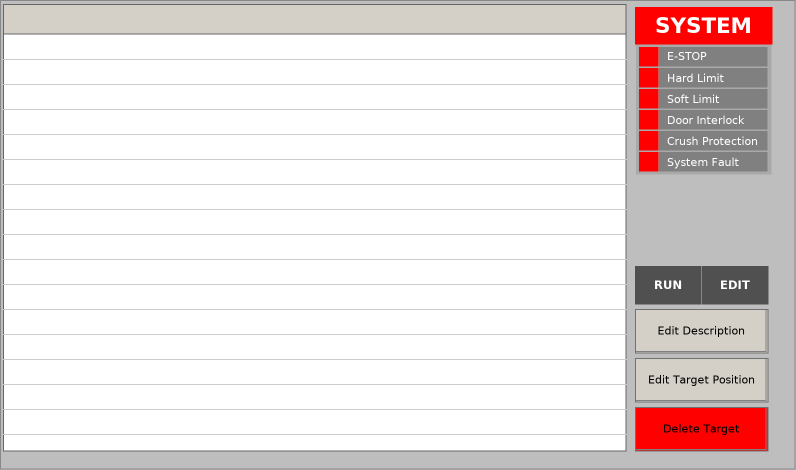
VISUALIZATION TARGET_PANEL  // 796x470
    Button (635,358 133x44), "Edit Target Position", colour toggle: (GV_HMI.ColorToggle[2])<>0, invisible if: HMI.bEditEnable<>1
        tap GV_HMI.ColorToggle[2]
        OnDialogClosed: execute {
            IF XML.savedvalues.savedpos[GV_HMI.RowSelect].target <= XML.savedvalues.UpSoftLim AND XML.savedvalues.savedpos[GV_HMI.RowSelect].target >= XML.savedvalues.DownSoftLim THEN
            	XML.savedvalues.savedpos[GV_HMI.RowSelect].targetclear := TRUE;
            ELSE
            	XML.savedvalues.savedpos[GV_HMI.RowSelect].targetclear := FALSE;
            END_IF
        }
        OnMouseDown: write XML.savedvalues.savedpos[.GV_HMI.RowSelect].target via VisuDialogs.Numpad, min XML.savedvalues.DownSoftLim, max XML.savedvalues.UpSoftLim, title 'Target Position'
    Button (635,309 133x44), "Edit Description", colour toggle: GV_HMI.ColorToggle[3], invisible if: HMI.bEditEnable<>1
        tap GV_HMI.ColorToggle[3]
        OnMouseDown: write XML.savedvalues.savedpos[.GV_HMI.RowSelect].description via VisuDialogs.Keypad
        OnMouseDown: execute {
            IF XML.savedvalues.savedpos[GV_HMI.RowSelect].target <= XML.savedvalues.UpSoftLim AND XML.savedvalues.savedpos[GV_HMI.RowSelect].target >= XML.savedvalues.DownSoftLim THEN
            	XML.savedvalues.savedpos[GV_HMI.RowSelect].targetclear := TRUE;
            ELSE
            	XML.savedvalues.savedpos[GV_HMI.RowSelect].targetclear := FALSE;
            END_IF
        }
    Table (3,4 623x447), data array: HMI.displayvalues
        p1420305297: GV_HMI.ColumnSelect
        p1137915858: GV_HMI.RowSelect
        p3854506369: HMI.displayvalues[INDEX].target
        p1892666644: HMI.displayvalues[INDEX].description
        p2232123230: Target Position
        p511219082: Description
    Rectangle (636,27 135x147)
    RoundedRectangle (639,47 19x19), colour toggle: GV_LIFT.ESTOP_INDICATOR_OUT
    RoundedRectangle (639,68 19x19), colour variable: HMI_Hard_Limits.HardLimitFlag
    RoundedRectangle (639,89 19x19), colour toggle: HMI.bSoftLimFlag
    RoundedRectangle (639,110 19x19), colour variable: HMI_Door_Toggle.dwDoorFlag
    RoundedRectangle (635,7 137x37), "SYSTEM", colour toggle: HMI_System_Indicator.bSystemFlag
    RoundedRectangle (639,131 19x19), colour variable: HMI_Crush_Indicator.dwCrushFlag
    RoundedRectangle (639,152 19x19), colour toggle: GV_LIFT.SYSTEM_FAULT <>1
    Rectangle (659,47 108x19)
    Rectangle (664,44 100x25), "E-STOP"
    Rectangle (659,68 108x19)
    Rectangle (664,66 100x25), "Hard Limit"
    Rectangle (659,89 108x19)
    Rectangle (664,87 100x25), "Soft Limit"
    Rectangle (659,110 108x19)
    Rectangle (664,108 100x25), "Door Interlock"
    Rectangle (659,131 108x19)
    Rectangle (664,129 100x25), "Crush Protection"
    Rectangle (659,152 108x19)
    Rectangle (664,150 100x25), "System Fault"
    Button (635,407 133x44), "Delete Target", colour toggle: (GV_HMI.ColorToggle[1])<>0, invisible if: HMI.bEditEnable<>1
        tap GV_HMI.ColorToggle[1]
        OnMouseDown: execute {
            XML.savedvalues.savedpos[GV_HMI.RowSelect].targetclear := FALSE;
            XML.savedvalues.savedpos[GV_HMI.RowSelect].target := 0.00;
            XML.savedvalues.savedpos[GV_HMI.RowSelect].description := '';
        }
    Rectangle (635,266 66x38), "RUN", colour toggle: HMI.bEditEnable<>0
        OnMouseDown: execute { HMI.bEditEnable:=FALSE; }
    Rectangle (702,266 66x38), "EDIT", colour toggle: HMI.bEditEnable<>1
        OnMouseDown: execute { HMI.bEditEnable:=TRUE; }
END_VISUALIZATION

(* stored: Version 1.1.0.1, ProductVersion 3.1.4022.12
   Visu TARGET_PANEL: Id {1dee17ff-8979-4ad8-a29f-7cc83dd1c9c4} *)
